PROGRAM MAIN
VAR
    ToggleAllRelaysFB : FB_ToggleRelays;
    ToggleAllRelaysButton : BOOL;              // HMI toggle button
    LastToggleState: BOOL;
    ToggleRelaysWithDelayButton : BOOL;        // HMI Button
    DelayedToggle : ToggleRelaysWithDelay;     // FB Instance
    Delay : TIME;                              // TIME type, gets converted from INT
    DelayMsInput : INT;                        // User input in ms from HMI
END_VAR


// Call function block for delayed toggle
DelayedToggle(
    StartDelayToggle := ToggleRelaysWithDelayButton,
    DelayMsInput := DelayMsInput,              // Directly pass the INT to FB
    BoolRelayArray := BoolRelayArray
);

// Call function block for instant toggle
ToggleAllRelaysFB(
    ToggleButton := ToggleAllRelaysButton,
    RelayArray := BoolRelayArray
);

END_PROGRAM

(* stored: Version 1.1.0.1, ProductVersion 3.1.4024.13
   POU MAIN: Id {63904485-10c2-4552-8766-9ea490077c86}, SpecialFunc None *)
